# EPICS substitutions: db/Beckhoff_7XXX/ecmcEL7411_CSP.substitutions
file "ecmcEL72XX_DRV_CSP.template"
{
  pattern {CH_ID}
          {01   }}
}

file "ecmcEL72XX_ENC.template"
{
  pattern {LINR,    ESLO,   EOFF,   EGU,        PREC, LOW, LOLO, HIGH, HIHI, HYST, LLSV,       LSV,        HSV,        HHSV      }
          {"SLOPE", 1,      0,      "Raw",      0,    0,   0,    0,    0,    0,    "NO_ALARM", "NO_ALARM", "NO_ALARM", "NO_ALARM"}
}
